PROGRAM FirstScan
VAR
	SkipFirstScan : BOOL; // You guessed it, this skips the after first scan!
END_VAR

IF SkipFirstScan = FALSE THEN
	
	//Default values for Ventalation
	Ventilation.SettingsArray[2].SpeedSetpointLow 	:= 3000;
	Ventilation.SettingsArray[1].SpeedSetpointLow 	:= 3000;
	Ventilation.SettingsArray[2].SpeedSetpointHigh 	:= 6000;
	Ventilation.SettingsArray[1].SpeedSetpointHigh 	:= 6000;
	
	
	
	SkipFirstScan := TRUE; // keep at bottom
	
END_IF

END_PROGRAM

(* stored: Version 1.1.0.1, ProductVersion 3.1.4024.12
   POU FirstScan: Id {683fc16c-20e6-46fc-9410-100e55b17f2b}, SpecialFunc None *)
